FUNCTION_BLOCK integEC (* Basic Function Block Type *)
  (* Standard: 61499-2 *)
  (* Version 0.0, 2007-06-14, milos, nxtControl GmbH, Template *)
  PACKAGE Main;
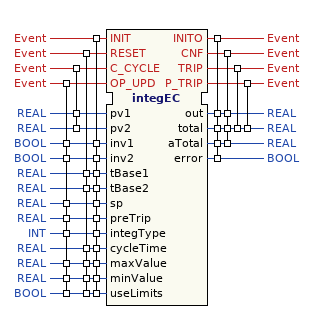
  EVENT_INPUT
    INIT WITH inv1, inv2, tBase1, tBase2, sp, preTrip, integType, cycleTime, maxValue, minValue, useLimits; (* Initialization Request *)
    RESET WITH tBase1, tBase2, cycleTime, maxValue, minValue, useLimits; (* reset integrator *)
    C_CYCLE WITH pv1, pv2; (* cycle calculation call *)
    OP_UPD WITH sp, preTrip, inv1, inv2, integType, maxValue, minValue, useLimits; (* new operator parameter *)
  END_EVENT
  EVENT_OUTPUT
    INITO WITH out, total, aTotal, error; (* Initialization Confirm *)
    CNF WITH out, total, aTotal; (* Execution Confirmation *)
    TRIP WITH total; (* total > sp *)
    P_TRIP WITH total; (* total > (sp - preTrip) *)
  END_EVENT
  VAR_INPUT
    pv1 : REAL := 0.0; (* pv1 to integrate *)
    pv2 : REAL := 0.0; (* pv2 to integrate *)
    inv1 : BOOL := FALSE; (* invert (multiply with -1) pv1 *)
    inv2 : BOOL := FALSE; (* invert (multiply with -1) pv2 *)
    tBase1 : REAL := 3600.0; (* timebase of pv1 [s] *)
    tBase2 : REAL := 3600.0; (* timebase of pv2 [s] *)
    sp : REAL := 0.0; (* setpoint of integrator *)
    preTrip : REAL := 0.0; (* distance to setpoint for preTrip to set *)
    integType : INT := 0; (* integration Type *)
    cycleTime : REAL := 1.0; (* cycle Time for calculation *)
    maxValue : REAL;
    minValue : REAL;
    useLimits : BOOL;
  END_VAR
  VAR_OUTPUT
    out : REAL := 0.0; (* out value (depends on integType) *)
    total : REAL := 0.0; (* integrated summation of all pv *)
    aTotal : REAL := 0.0; (* integrated summation of all ABS(pv) *)
    error : BOOL := FALSE; (* error detected *)
  END_VAR
  VAR
    sumPv : REAL := 0.0; (* time based sum of pv (with inv correction) *)
  END_VAR
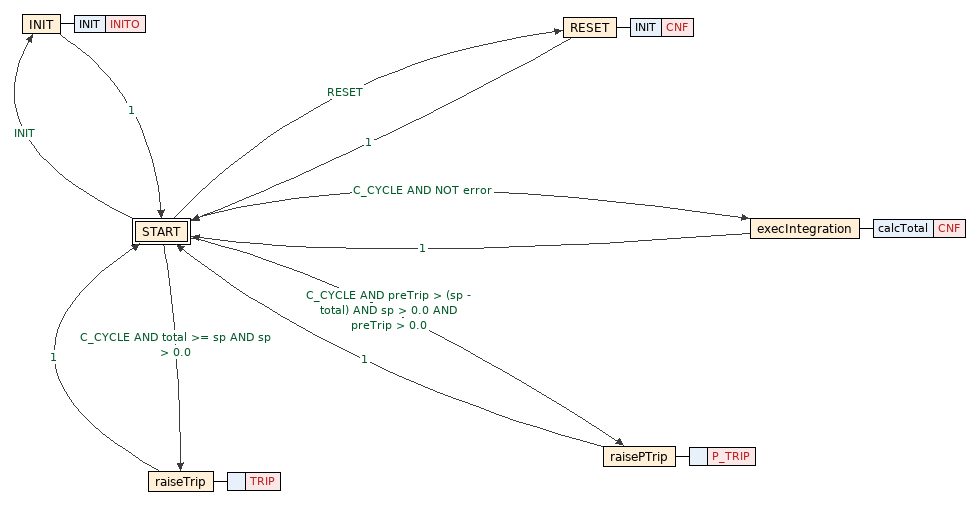
  EC_STATES
    START; (* Initial State *)
    INIT : INIT -> INITO; (* Initialization *)
    execIntegration : calcTotal -> CNF; (* Normal execution *)
    raiseTrip : -> TRIP;
    raisePTrip : -> P_TRIP;
    RESET : INIT -> CNF;
  END_STATES
  EC_TRANSITIONS
    START TO INIT := INIT;
    INIT TO START := 1;
    START TO execIntegration := C_CYCLE AND NOT error;
    execIntegration TO START := 1;
    START TO raiseTrip := C_CYCLE AND total >= sp AND sp > 0.0;
    START TO raisePTrip := C_CYCLE AND preTrip > (sp - total) AND sp > 0.0 AND preTrip > 0.0;
    raisePTrip TO START := 1;
    raiseTrip TO START := 1;
    START TO RESET := RESET;
    RESET TO START := 1;
  END_TRANSITIONS
  ALGORITHM INIT IN ST: (* Initialization algorithm *)
out := 30.0;
total := 30.0;
aTotal := 30.0;
error := (tBase1 <= 0.0) OR (tBase2 <= 0.0) OR (cycleTime <= 0.0);
  END_ALGORITHM
  ALGORITHM calcTotal IN ST:
aTotal := aTotal + cycleTime * (pv1/tBase1 + pv2/tBase2);

IF inv1 THEN
 sumPv := pv1/tBase1 * -1;
ELSE
 sumPv := pv1/tBase1;
END_IF;
IF inv2 THEN
 sumPv := sumPv + pv2/tBase2 * -1;
ELSE
 sumPv := sumPv + pv2/tBase2;
END_IF;

total := total + cycleTime * sumPv;

IF useLimits THEN
 total := LIMIT(minValue, total, maxValue);
END_IF;

IF integType = 1 AND sp > 0.0 THEN
 out := sp-total;
ELSE
 out := total;
END_IF;
  END_ALGORITHM
END_FUNCTION_BLOCK
